Staubli VAL3: Control_ListBS.pgx

public program Control_ListBS(string x_sItemName, string x_sItemValue, num x_nSelectItem, num x_nText)
  local string l_sBuff[10]
  local string l_sValue[10]
  local num l_nIndex
  local bool l_bRes
begin
    //说明：
  //函数功能：在划定的框内，把选中项给显示出来
  //l_nFirst  在列表中第一个显示的项的序号
  //x_nSelectItem  被选中的项的序号
  //l_nCount 合法列表项的项总数，如何数组中间为空，则可能被截断

   // 赋初值
   for l_nIndex=0 to size(l_sBuff)-1
    l_sBuff[l_nIndex]=""
  endFor

  //把项的名字给解析出来
  call  Str_SplitComma(l_bRes,x_sItemName,l_sBuff)
  if !l_bRes
    return
  endIf

    call  Str_SplitComma(l_bRes,x_sItemValue,l_sValue)
  if !l_bRes
    return
  endIf

  call Control_PanelXY(nPanelLTopX,nPanelLTopY,nPanelWidthX/2,nPanelLengthY)
  call Control_List(l_sBuff,x_nSelectItem)
  call Control_PanelXY(nPanelLTopX+nPanelWidthX/2,nPanelLTopY,nPanelWidthX/2,nPanelLengthY)
  call Control_List(l_sValue,x_nSelectItem)

end
